// LS Electric XG5000 project: 실린더2
// PLC LSPLC

PROGRAM NewProgram (task: 스캔 프로그램)

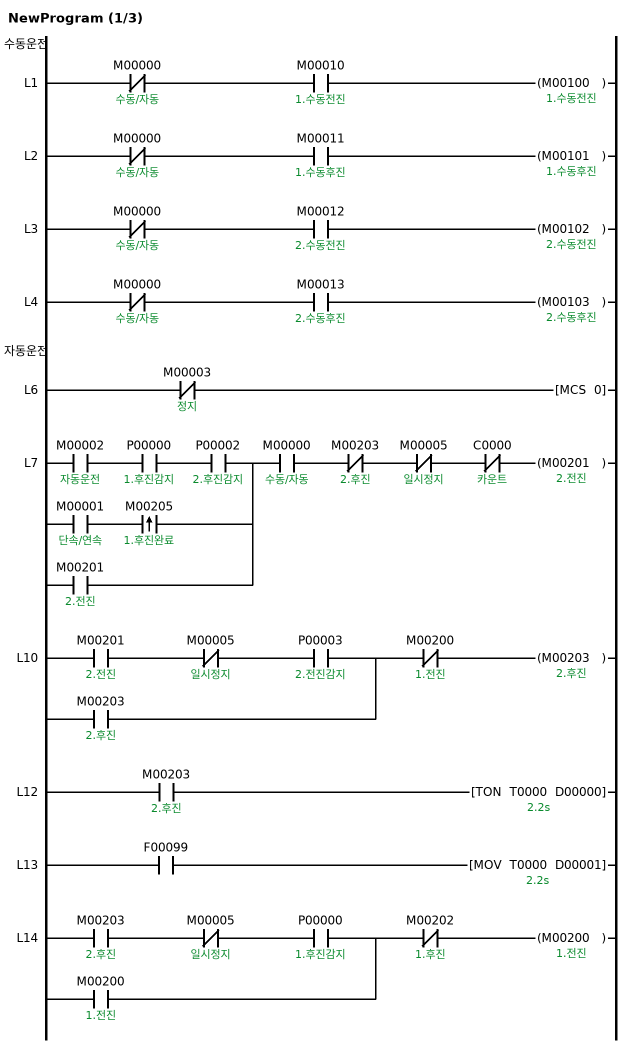
수동운전:
; L1
LOAD NOT  M00000	// 수동/자동
AND       M00010	// 1.수동전진
OUT       M00100	// 1.수동전진
; L2
LOAD NOT  M00000	// 수동/자동
AND       M00011	// 1.수동후진
OUT       M00101	// 1.수동후진
; L3
LOAD NOT  M00000	// 수동/자동
AND       M00012	// 2.수동전진
OUT       M00102	// 2.수동전진
; L4
LOAD NOT  M00000	// 수동/자동
AND       M00013	// 2.수동후진
OUT       M00103	// 2.수동후진
자동운전:
; L6
LOAD NOT  M00003	// 정지
MCS       0
; L7
LOAD      M00002	// 자동운전
AND       P00000	// 1.후진감지
AND       P00002	// 2.후진감지
LOAD      M00001	// 단속/연속
ANDP      M00205	// 1.후진완료
OR LOAD
OR        M00201	// 2.전진
AND       M00000	// 수동/자동
AND NOT   M00203	// 2.후진
AND NOT   M00005	// 일시정지
AND NOT   C0000	// 카운트
OUT       M00201	// 2.전진
; L10
LOAD      M00201	// 2.전진
AND NOT   M00005	// 일시정지
AND       P00003	// 2.전진감지
OR        M00203	// 2.후진
AND NOT   M00200	// 1.전진
OUT       M00203	// 2.후진
; L12
LOAD      M00203	// 2.후진
TON       T0000 D00000	// 2.2s
; L13
LOAD      F00099
MOV       T0000 D00001	// 2.2s
; L14
LOAD      M00203	// 2.후진
AND NOT   M00005	// 일시정지
AND       P00000	// 1.후진감지
OR        M00200	// 1.전진
AND NOT   M00202	// 1.후진
OUT       M00200	// 1.전진

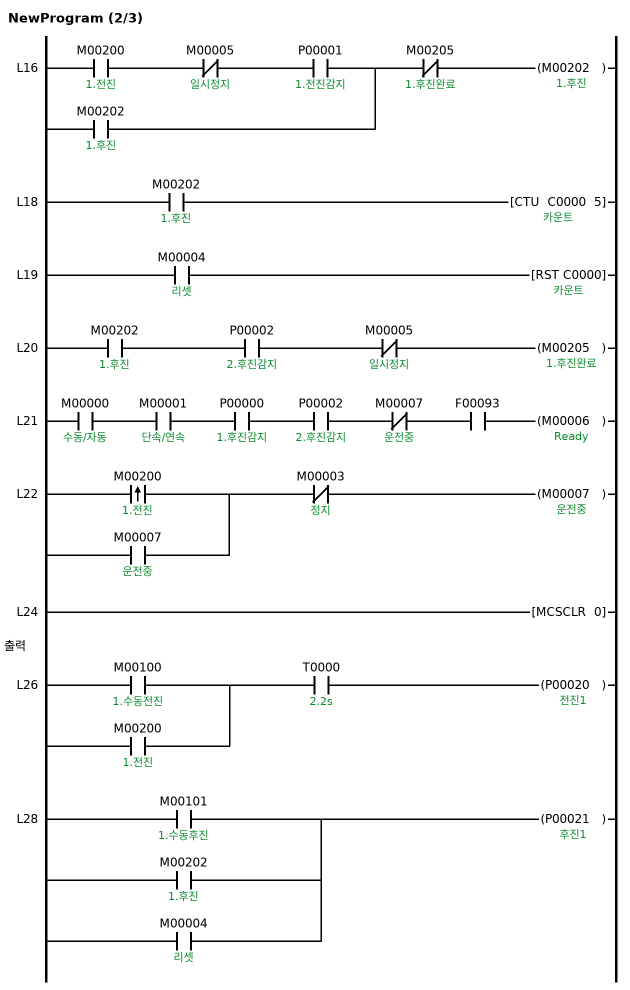
; L16
LOAD      M00200	// 1.전진
AND NOT   M00005	// 일시정지
AND       P00001	// 1.전진감지
OR        M00202	// 1.후진
AND NOT   M00205	// 1.후진완료
OUT       M00202	// 1.후진
; L18
LOAD      M00202	// 1.후진
CTU       C0000 5	// 카운트
; L19
LOAD      M00004	// 리셋
RST       C0000	// 카운트
; L20
LOAD      M00202	// 1.후진
AND       P00002	// 2.후진감지
AND NOT   M00005	// 일시정지
OUT       M00205	// 1.후진완료
; L21
LOAD      M00000	// 수동/자동
AND       M00001	// 단속/연속
AND       P00000	// 1.후진감지
AND       P00002	// 2.후진감지
AND NOT   M00007	// 운전중
AND       F00093
OUT       M00006	// Ready
; L22
LOADP     M00200	// 1.전진
OR        M00007	// 운전중
AND NOT   M00003	// 정지
OUT       M00007	// 운전중
; L24
MCSCLR    0
출력:
; L26
LOAD      M00100	// 1.수동전진
OR        M00200	// 1.전진
AND       T0000	// 2.2s
OUT       P00020	// 전진1
; L28
LOAD      M00101	// 1.수동후진
OR        M00202	// 1.후진
OR        M00004	// 리셋
OUT       P00021	// 후진1

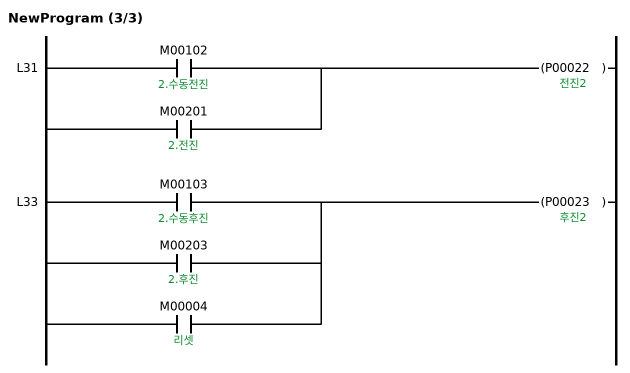
; L31
LOAD      M00102	// 2.수동전진
OR        M00201	// 2.전진
OUT       P00022	// 전진2
; L33
LOAD      M00103	// 2.수동후진
OR        M00203	// 2.후진
OR        M00004	// 리셋
OUT       P00023	// 후진2

VARIABLES AND COMMENTS (devices not used above)
M00204	BIT	2.후진완료